PROGRAM Mode
VAR
	AutoModePB: BOOL;
	ManualModePB: BOOL;
	AutoMode: BOOL;
	ManualMode: BOOL;
	Off: BOOL;
	Mode1PB: BOOL;
	Mode1: BOOL;
	Mode2PB: BOOL;
	Mode3PB: BOOL;
	OffPB: BOOL;
	Mode2: BOOL;
END_VAR


VAR_INPUT
	Mode3: BOOL;
END_VAR

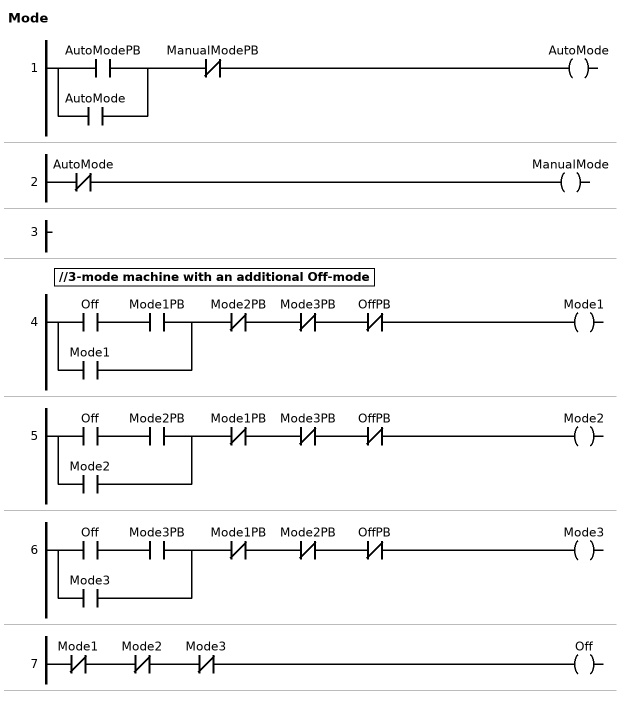
// NETWORK 1
AutoMode := (AutoModePB OR AutoMode) AND NOT ManualModePB;

// NETWORK 2
ManualMode := NOT AutoMode;

// NETWORK 3

// NETWORK 4
// label: //3-mode machine with an additional Off-mode
Mode1 := (Off AND Mode1PB OR Mode1) AND NOT Mode2PB AND NOT Mode3PB AND NOT OffPB;

// NETWORK 5
Mode2 := (Off AND Mode2PB OR Mode2) AND NOT Mode1PB AND NOT Mode3PB AND NOT OffPB;

// NETWORK 6
Mode3 := (Off AND Mode3PB OR Mode3) AND NOT Mode1PB AND NOT Mode2PB AND NOT OffPB;

// NETWORK 7
Off := NOT Mode1 AND NOT Mode2 AND NOT Mode3;

END_PROGRAM

(* stored: Version 1.1.0.1, ProductVersion 3.1.4024.10
   POU Mode: Id {462bcb6b-eaac-4e7c-8128-9b8ca43a24e1}, SpecialFunc None *)
